(* PLC project Unnamed, Unknown Unnamed 1 *)
(* stored: creationDateTime 2025-12-15T22:21:58, modificationDateTime 2025-12-15T23:38:39 *)

PROGRAM program4
  VAR
    Reset_Btn AT %IX0.2 : BOOL;
    Count_Btn AT %IX0.1 : BOOL;
    LED AT %QX0.1 : BOOL;
  END_VAR
  VAR
    Counter1 : CTU;
    Count_Edge : R_TRIG;
  END_VAR
  VAR CONSTANT
    Preset : INT := 5;
  END_VAR
  VAR  (* added by the conversion: wires and edge detectors of the diagram *)
    R_TRIG1 : R_TRIG;
  END_VAR

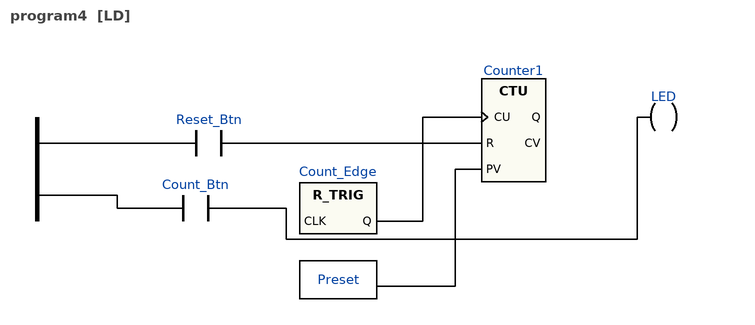
(* LD diagram, written out as Structured Text *)
LED := Count_Btn;
Count_Edge();
R_TRIG1(CLK := Count_Edge.Q);
Counter1(CU := R_TRIG1.Q, R := Reset_Btn, PV := Preset);
END_PROGRAM

CONFIGURATION Config0
  RESOURCE Res0 ON PLC
    TASK task0(INTERVAL := T#20ms, PRIORITY := 0);
    PROGRAM instance0 WITH task0 : program4;
  END_RESOURCE
END_CONFIGURATION
